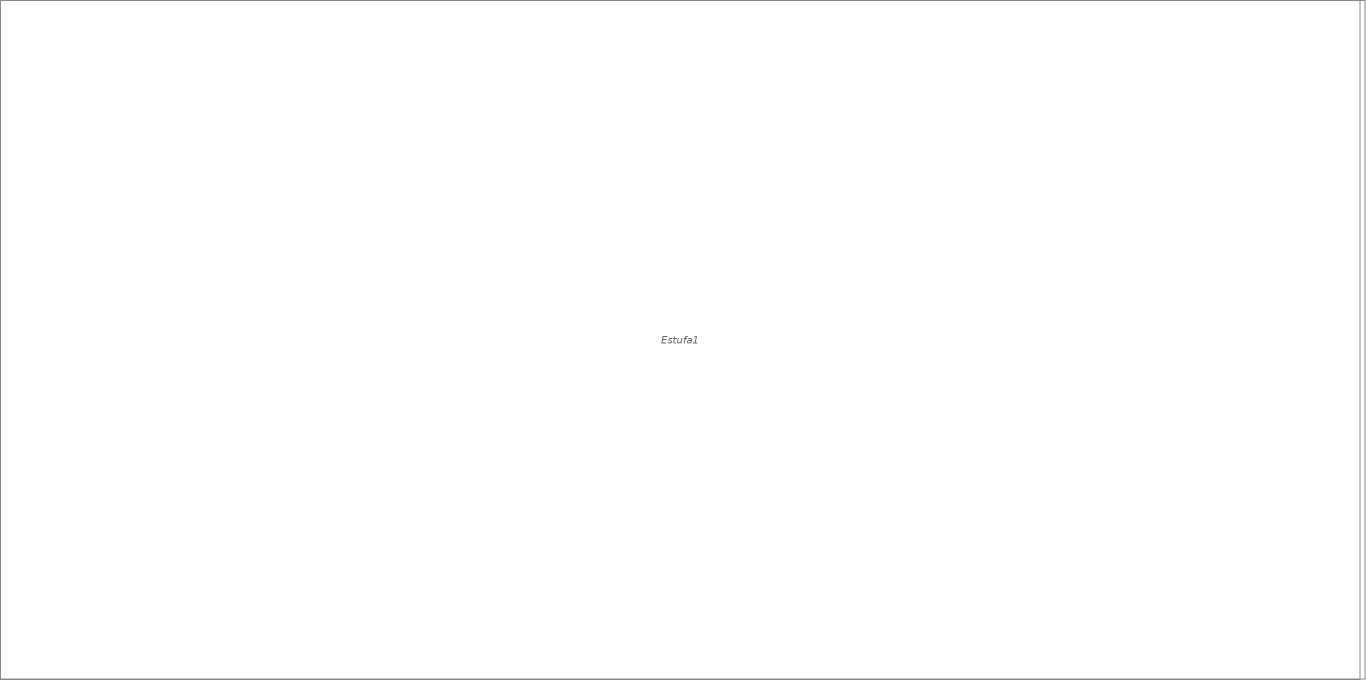
VISUALIZATION Aba_Estufa  // 1366x680
    TabControl (0,0 1360x680)
        shows Estufa1()
        shows Grafico()
        [0]: TabTitle=Dashboard
        [1]: TabTitle=Gráfico
END_VISUALIZATION

(* stored: Version 1.1.0.1, ProductVersion 3.1.4024.12
   Visu Aba_Estufa: Id {1293aca4-a602-4352-95f1-5f64cd4003a8} *)
